Staubli VAL3: stop_print.pgx

public program stop_print()
begin

      // arrêt pompe
    dioSet(doPompe,0)
    put("Pompe arret")
      // fermeture obturateur
    dioSet(doValve2,0)
    dioSet(doValve1,1)
    put("Obturateur ferme")

end
